Staubli VAL3: Day1.dtx

num nVector[10]
num nResult
string sInput
num nResult2
bool bResult
num nInput
